FUNCTION ArgToIBinArg : Result
VAR_INPUT
	iArg		: I_Arg;
END_VAR
VAR_OUTPUT
	iVal		: I_BinArg;
END_VAR

IF __QUERYINTERFACE(iArg, iVal) THEN
	ArgToIBinArg := Ok;
END_IF

END_FUNCTION

(* stored: Version 1.1.0.1
   POU ArgToIBinArg: Id {251bbc86-8ca7-4831-8a1b-2f5e6a418da8}, SpecialFunc None *)
